// TIA Portal V20 export
VAR_GLOBAL   // PLC tag table "Constantes del Router"
   Estado_Inicializacion_1 AT %M50.0 : Bool;
   Estado_Inicializacion_2 AT %M50.1 : Bool;
   Estado_Inicializacion_3 AT %M50.2 : Bool;
   Estado_Inicializacion_4 AT %M50.3 : Bool;
   Estado_Inicializacion_5 AT %M50.4 : Bool;
   Estado_Inicializacion_6 AT %M50.5 : Bool;
   Estado_Inicializacion_7 AT %M50.6 : Bool;
   Estado_Inicializacion_8 AT %M50.7 : Bool;
   Mem_Actual_JDT1_INIR_1 AT %M51.0 : Bool;
   Mem_Actual_JDT1_INIR_2 AT %M51.1 : Bool;
   Mem_Actual_JDT1_INIR_3 AT %M51.2 : Bool;
   Mem_Actual_JDT1_INIR_4 AT %M51.3 : Bool;
   Mem_Actual_JDT1_INIR_5 AT %M51.4 : Bool;
   Mem_Actual_JDT1_INIR_6 AT %M51.5 : Bool;
   Mem_Actual_JDT1_INIR_7 AT %M51.6 : Bool;
   Mem_Actual_JDT1_INIR_8 AT %M51.7 : Bool;
   Mem_Actual_JDT2_INIR_1 AT %M52.0 : Bool;
   Mem_Actual_JDT2_INIR_2 AT %M52.1 : Bool;
   Mem_Actual_JDT2_INIR_3 AT %M52.2 : Bool;
   Mem_Actual_JDT2_INIR_4 AT %M52.3 : Bool;
   Mem_Actual_JDT2_INIR_5 AT %M52.4 : Bool;
   Mem_Actual_JDT2_INIR_6 AT %M52.5 : Bool;
   Mem_Actual_JDT2_INIR_7 AT %M52.6 : Bool;
   Mem_Actual_JDT2_INIR_8 AT %M52.7 : Bool;
   Refresco_INIR_JDT01 AT %MB51 : Byte;
   Refresco_INIR_JDT02 AT %MB52 : Byte;
   Estado_inicializacion AT %MB50 : Byte;
END_VAR
VAR_GLOBAL CONSTANT   // user constants
   ROUT_Cantidad_Etiquetas_DB : UInt := 1000;   // Numero máximo de etiquetas almacenadas en cada DB de etiquetas
   ROUT_CaracterRelleno : Byte := '0';   // caracter de relleno para alfanumerico
   ROUT_Long_Dat_Scanner : UInt := 34;   // Longitud Datos Entrada/Salida de cada Scanner (Bytes)
   ROUT_Long_Etiqueta : UInt := 20;   // Caracteres de la etiqueta Fisica + 1 ('N'+'123456789')
   ROUT_Long_Reg_Datos_Etiqueta : UInt := 12;   // Longitud del registro de bits de cruces expresado en bytes (MAX:12)
   ROUT_Long_Reg_Datos_FIFO : UInt := 10;   // Longitud en Bytes de los datos de una orden en la fifo
   ROUT_Max_Destinos : UInt := 100;   // número máximo de destinos presentes en la instalación. siempre tener en cuenta todos los destinos incluso los que no sean del mismo PLC
   ROUT_Max_Lec_Ciclo : UInt := 26;   // Numero maximo de lecturas de scanner que se tratan en un ciclo de SCAN
   ROUT_Max_Reg_Etiquetas : UInt := 4000;   // Numero maximo de etiquetas permitidas en los DB de datos
   ROUT_Max_Scanners : UInt := 199;   // numero máximo de scanners en la instalación. tamaño del ROUT_NDB_Lectura_SCR
   ROUT_N_Colas : UInt := 10000;   // Número de Colas
   ROUT_NDB_Etiquetas_Esp : UInt := 209;   // Numero de DB de Etiquetas Especiales
   ROUT_NDB_FIFO_Odr_SCR : UInt := 213;   // Numero de DB donde se extraen las ordenes de los scanners a la fifo
   ROUT_NDB_Ini_Reg_Etiq : UInt := 201;   // Numero de DB donde empiezan los registros de etiquetas. Cuidado, el resto de registros va en números consecutivos
   ROUT_NDB_Lectura_SCR : UInt := 211;   // Numero de DB donde se guardan las lecturas recogidas de los scanners.
   ROUT_Num_Max_Desvios : UInt := 20;   // número máximo de desvios presentes en una ruta de una instalacion
   ROUT_Num_Ordenes_FIFO : UInt := 1;   // Numero de ordenes que se pueden quardar en la Fifo de un scanner
   ROUT_NDB_FIFO_ORDENES_S2 : UInt := 220;
   ROUT_LONG_FIFO_ORDENES_S2 : UInt := 5;
   ROUT_NDB_FIFO_ORDENES_S3 : UInt := 221;
   ROUT_LONG_FIFO_ORDENES_S3 : UInt := 5;
   ROUT_NDB_FIFO_ORDENES_S4 : UInt := 222;
   ROUT_LONG_FIFO_ORDENES_S4 : UInt := 5;
   ROUT_NDB_Tipo_Scanner : UInt := 912;
   ROUT_NDB_Cola_Etiqueta : UInt := 212;
   ROUT_Long_Reg_Datos_Caja : UInt := 10;
   ROUT_DB_Eventos_Router : Word := 210;
   ROUT_X_CONEX_JDT1 : Bool := TRUE;   // TRUE conexion principal, false secundaria
   con_sello_tiempo : Bool := true;
END_VAR
